{attribute 'qualified_only'}
{attribute 'strict'}
TYPE EControlModePiano450 :
(
	PowerMode
);
END_TYPE

(* stored: Version 1.1.0.1, ProductVersion 3.1.4024.4
   DUT EControlModePiano450: Id {449ef594-84cd-4b67-bc62-96ca0d33efc3} *)
